// SIMATIC STEP 7 (V5.x) project Q5
// CPU: CPU 313C
// station: Hardware
// station: SIMATIC 300(1)
// station: P_ADR_BUS
// program: S7 Program(1)

SYMBOL_TABLE
"Box Counter"	C 0	COUNTER
"Rotation Counter"	C 2	COUNTER
"X Counter"	C 3	COUNTER
"Z Counter"	C 4	COUNTER
"Cycle Counter"	C 5	COUNTER
"Out put Counter"	C 6	COUNTER
"Start"	I 0.0	BOOL
"Stop"	I 0.1	BOOL
"Reset Counter"	I 0.2	BOOL
"Pallet Sensor"	I 0.3	BOOL
"Box Sensor"	I 0.4	BOOL
"Moving-X"	I 0.6	BOOL
"Moving-Z"	I 0.7	BOOL
"Rotating"	I 1.0	BOOL
"Force stop"	I 2.0	BOOL
"Start/Stop mem"	M 0.0	BOOL
"Memory Pallet"	M 0.1	BOOL
"Memory Box"	M 0.2	BOOL
"RisingEdge pallet sens"	M 0.3	BOOL
"RisingEdge pallet mem"	M 0.4	BOOL
"RisingEdge Box sens"	M 0.5	BOOL
"RisingEdge Box mem"	M 0.6	BOOL
"RisingEdge COUNT ROTATE"	M 3.0	BOOL
"RisingEdge COUNT X"	M 3.1	BOOL
"RisingEdge COUNT Z"	M 3.2	BOOL
"RisingEdge COUNT BOX"	M 3.3	BOOL
"Box-count"	MW 10	WORD
"Cycle-count"	MW 15	WORD
"Rotate-Move-count"	MW 20	WORD
"X-Move-count"	MW 25	WORD
"Z-Move-count"	MW 30	WORD
"Start Button"	Q 0.0	BOOL
"Stop Button"	Q 0.1	BOOL
"Reset Button"	Q 0.2	BOOL
"Pallet Coneyor"	Q 0.3	BOOL
"Box Conveyor"	Q 0.4	BOOL
"X Out"	Q 0.5	BOOL
"Z Out"	Q 0.6	BOOL
"CW Out"	Q 0.7	BOOL
"CCW Out"	Q 1.0	BOOL
"Grab"	Q 1.1	BOOL
"Output"	QD 30	DWORD
"Delay Box sensor"	T 0	TIMER
END_SYMBOL_TABLE

ORGANIZATION_BLOCK OB 1
TITLE = "Main Program Sweep (Cycle)"
VERSION : 0.1
VAR_TEMP
  OB1_EV_CLASS : BYTE ;	//Bits 0-3 = 1 (Coming event), Bits 4-7 = 1 (Event class 1)
  OB1_SCAN_1 : BYTE ;	//1 (Cold restart scan 1 of OB 1), 3 (Scan 2-n of OB 1)
  OB1_PRIORITY : BYTE ;	//Priority of OB Execution
  OB1_OB_NUMBR : BYTE ;	//1 (Organization block 1, OB1)
  OB1_RESERVED_1 : BYTE ;	//Reserved for system
  OB1_RESERVED_2 : BYTE ;	//Reserved for system
  OB1_PREV_CYCLE : INT ;	//Cycle time of previous OB1 scan (milliseconds)
  OB1_MIN_CYCLE : INT ;	//Minimum cycle time of OB1 (milliseconds)
  OB1_MAX_CYCLE : INT ;	//Maximum cycle time of OB1 (milliseconds)
  OB1_DATE_TIME : DATE_AND_TIME ;	//Date and time OB1 started
END_VAR
BEGIN
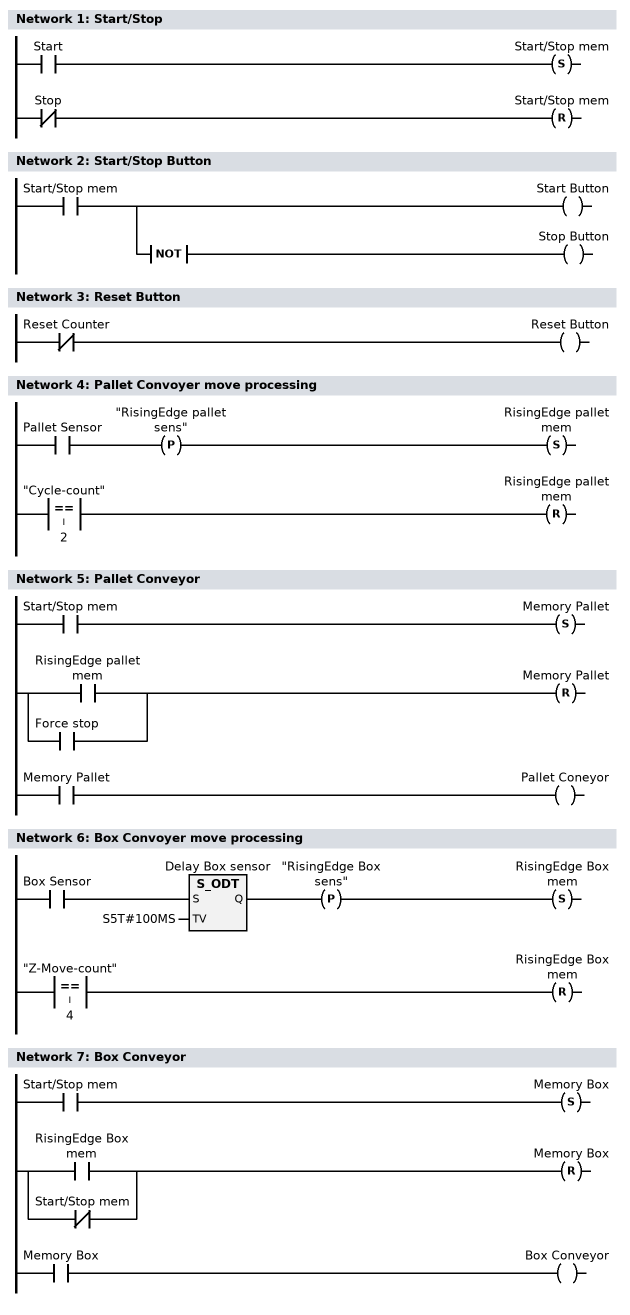
NETWORK
TITLE = Start/Stop
      A     "Start";
      S     "Start/Stop mem";
      AN    "Stop";
      R     "Start/Stop mem";
      NOP   0;
NETWORK
TITLE = Start/Stop Button
      A     "Start/Stop mem";
      =     L 20.0;
      A     L 20.0;
      BLD   102;
      =     "Start Button";
      A     L 20.0;
      NOT;
      =     "Stop Button";
NETWORK
TITLE = Reset Button
      AN    "Reset Counter";
      =     "Reset Button";
NETWORK
TITLE = Pallet Convoyer move processing
      A     "Pallet Sensor";
      FP    "RisingEdge pallet sens";
      S     "RisingEdge pallet mem";
      A(;
      L     "Cycle-count";
      L     2;
      ==I;
      );
      R     "RisingEdge pallet mem";
      NOP   0;
NETWORK
TITLE = Pallet Conveyor
      A     "Start/Stop mem";
      S     "Memory Pallet";
      A(;
      O     "RisingEdge pallet mem";
      O     "Force stop";
      );
      R     "Memory Pallet";
      A     "Memory Pallet";
      =     "Pallet Coneyor";
NETWORK
TITLE = Box Convoyer move processing
      A(;
      A     "Box Sensor";
      L     S5T#100MS;
      SD    "Delay Box sensor";
      NOP   0;
      NOP   0;
      NOP   0;
      A     "Delay Box sensor";
      );
      FP    "RisingEdge Box sens";
      S     "RisingEdge Box mem";
      A(;
      L     "Z-Move-count";
      L     4;
      ==I;
      );
      R     "RisingEdge Box mem";
      NOP   0;
NETWORK
TITLE = Box Conveyor
      A     "Start/Stop mem";
      S     "Memory Box";
      A(;
      O     "RisingEdge Box mem";
      ON    "Start/Stop mem";
      );
      R     "Memory Box";
      A     "Memory Box";
      =     "Box Conveyor";
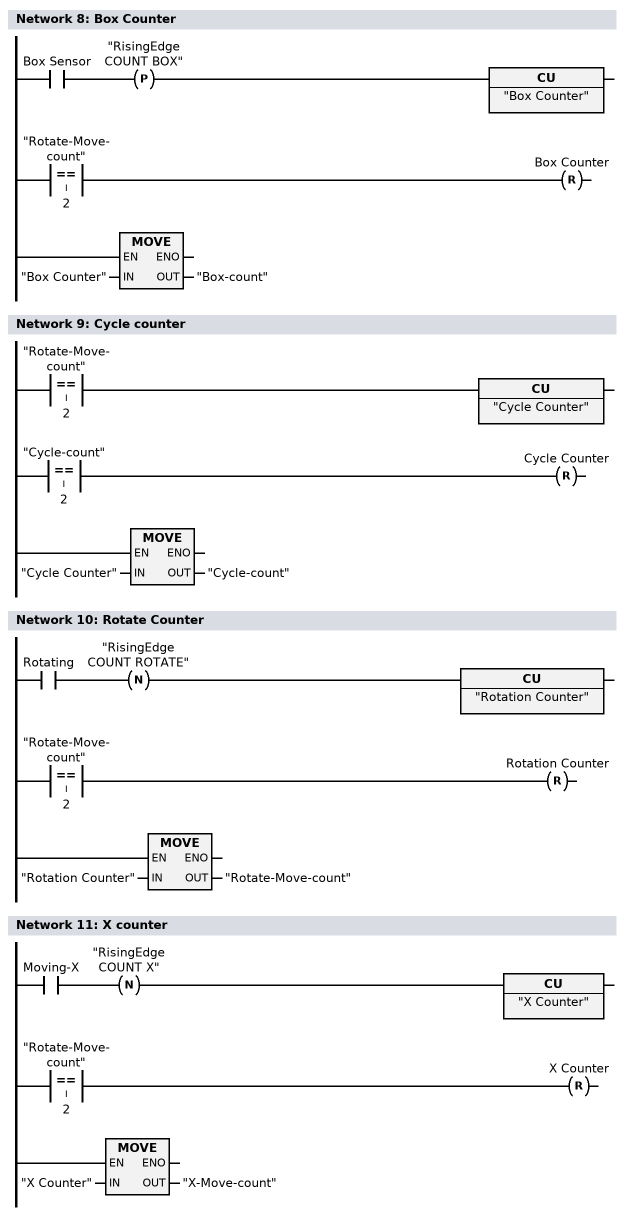
NETWORK
TITLE = Box Counter
      A     "Box Sensor";
      FP    "RisingEdge COUNT BOX";
      CU    "Box Counter";
      BLD   101;
      NOP   0;
      NOP   0;
      A(;
      L     "Rotate-Move-count";
      L     2;
      ==I;
      );
      R     "Box Counter";
      L     "Box Counter";
      T     "Box-count";
      NOP   0;
      NOP   0;
NETWORK
TITLE = Cycle counter
      A(;
      L     "Rotate-Move-count";
      L     2;
      ==I;
      );
      CU    "Cycle Counter";
      BLD   101;
      NOP   0;
      NOP   0;
      A(;
      L     "Cycle-count";
      L     2;
      ==I;
      );
      R     "Cycle Counter";
      L     "Cycle Counter";
      T     "Cycle-count";
      NOP   0;
      NOP   0;
NETWORK
TITLE = Rotate Counter
      A     "Rotating";
      FN    "RisingEdge COUNT ROTATE";
      CU    "Rotation Counter";
      BLD   101;
      NOP   0;
      NOP   0;
      A(;
      L     "Rotate-Move-count";
      L     2;
      ==I;
      );
      R     "Rotation Counter";
      L     "Rotation Counter";
      T     "Rotate-Move-count";
      NOP   0;
      NOP   0;
NETWORK
TITLE = X counter
      A     "Moving-X";
      FN    "RisingEdge COUNT X";
      CU    "X Counter";
      BLD   101;
      NOP   0;
      NOP   0;
      A(;
      L     "Rotate-Move-count";
      L     2;
      ==I;
      );
      R     "X Counter";
      L     "X Counter";
      T     "X-Move-count";
      NOP   0;
      NOP   0;
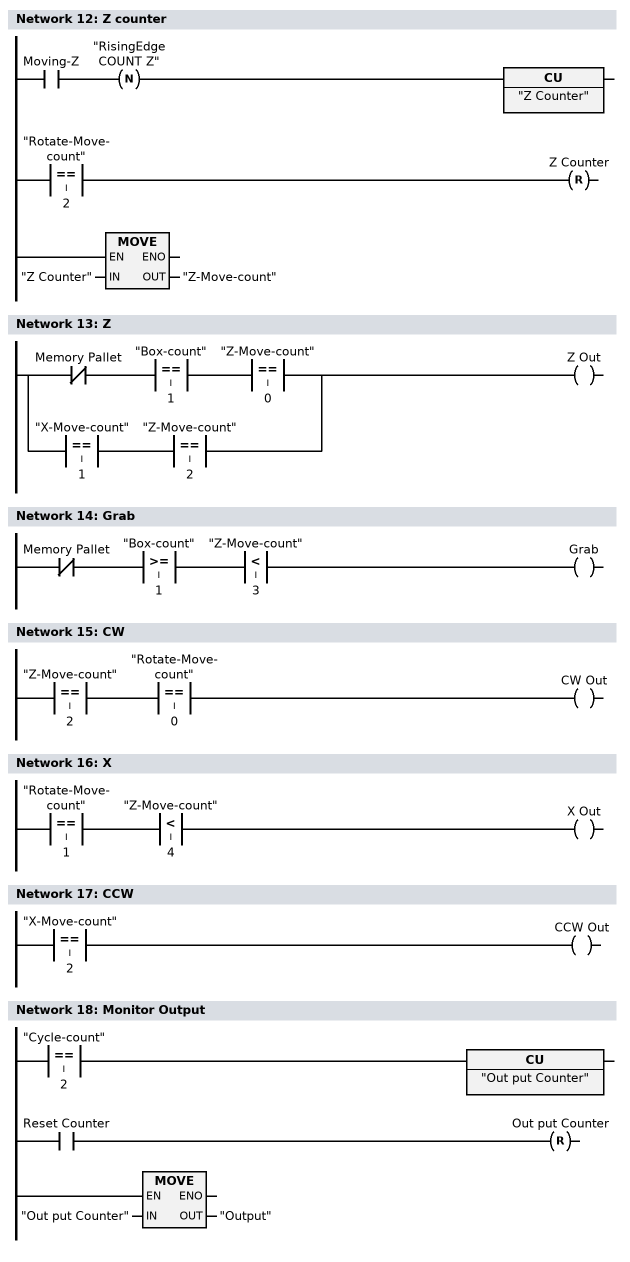
NETWORK
TITLE = Z counter
      A     "Moving-Z";
      FN    "RisingEdge COUNT Z";
      CU    "Z Counter";
      BLD   101;
      NOP   0;
      NOP   0;
      A(;
      L     "Rotate-Move-count";
      L     2;
      ==I;
      );
      R     "Z Counter";
      L     "Z Counter";
      T     "Z-Move-count";
      NOP   0;
      NOP   0;
NETWORK
TITLE = Z
      AN    "Memory Pallet";
      A(;
      L     "Box-count";
      L     1;
      ==I;
      );
      A(;
      L     "Z-Move-count";
      L     0;
      ==I;
      );
      O;
      A(;
      L     "X-Move-count";
      L     1;
      ==I;
      );
      A(;
      L     "Z-Move-count";
      L     2;
      ==I;
      );
      =     "Z Out";
NETWORK
TITLE = Grab
      AN    "Memory Pallet";
      A(;
      L     "Box-count";
      L     1;
      >=I;
      );
      A(;
      L     "Z-Move-count";
      L     3;
      <I;
      );
      =     "Grab";
NETWORK
TITLE = CW
      A(;
      L     "Z-Move-count";
      L     2;
      ==I;
      );
      A(;
      L     "Rotate-Move-count";
      L     0;
      ==I;
      );
      =     "CW Out";
NETWORK
TITLE = X
      A(;
      L     "Rotate-Move-count";
      L     1;
      ==I;
      );
      A(;
      L     "Z-Move-count";
      L     4;
      <I;
      );
      =     "X Out";
NETWORK
TITLE = CCW
      L     "X-Move-count";
      L     2;
      ==I;
      =     "CCW Out";
NETWORK
TITLE = Monitor Output
      A(;
      L     "Cycle-count";
      L     2;
      ==I;
      );
      CU    "Out put Counter";
      BLD   101;
      NOP   0;
      NOP   0;
      A     "Reset Counter";
      R     "Out put Counter";
      L     "Out put Counter";
      T     "Output";
      NOP   0;
      NOP   0;
END_ORGANIZATION_BLOCK
